Fanuc KAREL source: kt00735.KL

-- PROVISIONAL review KL for V1013-1; original PC SHA256 ca46ea4467234a8690c721f0733b9b8f4b56aeca80e838f9b449fc8eb42a5ad1
-- Incomplete behavior may be omitted. Consult companion uncertainty JSON. Do not deploy.
PROGRAM KT00735
%NOLOCKGROUP
VAR
  OUT : INTEGER
-- UNRESOLVED_DECL ARG type=002012
BEGIN
  -- UNRESOLVED_PC offsets 5-18; opcodes 22,1D,23
  -- UNRESOLVED_PC offsets 23-27; opcodes 7F
END KT00735
